	fbWriteSPLuxLevel				: SH_Light.FB_TwoVal_SelectOne_RTrigChange;
	fbWritePirDelayTIme			: SH_Light.FB_TwoVal_SelectOne_RTrigChange;
	stRoomDataPLC					: SH_Light.ST_RoomDataPLC	:=	(
																	uiPirOffDelayTime	:= 30,
																	uiSpLuxLevel			:= 500,
																	uiPirDimDelayTime	:= 15,
																	uiSpDimLuxLevel		:= 200);
																	
	fbBallastOnHours				: SH_Light.FB_CountOnHours;
	bEnableHourCount			: BOOL := TRUE;
	
	//Non-persistent modbus data
	bPirActive_MB				AT %MX40.0	: BOOL;				//bPirLys i gammel kode
	uiActLuxLevel_MB			AT %MB44	: UINT;				//intHMIAktueltLux i gammel kode
	uiActLightLevelPct_MB	    AT %MB52	: UINT;				//intDALI_Gruppe1_Lysniveau i gammel kode
	
	//For Conversion
	uiPirOffMinutes						: UINT;
	udTimeScaling						: UDINT := 60000;
	uiLuxOn								: UINT;
	
	//max values checks
	uiMaxLuxLevel						: UINT := 1023;
	uiMaxPirOffMinutes			    	: UINT := 180;

	
END_VAR

VAR CONSTANT
    Sensor_DALI_LINE_NUM				: BYTE := 3;
	DALI_LINE_NUM_LIGHT			    	: BYTE := 1;
	DALI_LINE_NUM_PENDANTS	            : BYTE := 1; //0=ingen pendler
	arrSensitivityOccupancy				: ARRAY[1..3] OF BYTE := [4,4,4];
END_VAR
VAR PERSISTENT
	stPirSensorData: SH_Light.ST_DALI_Sensor;
	stTuneData: SH_Light.ST_TuneData_EX;

	uiPirOffDelayTime_MB	AT %MB42	: UINT;				//ntHMI_Pir_SetValue i gammel kode
	uiSPLuxLevel_MB			AT %MB48	: UINT;				//intHMI_Lux_SetValue i gammel kode
	uiBallastOnHours_MB		AT %MB56	: UINT;				//dintHMILysbraendtimer1 i gammel kode
	byOnHoursOverflowCount				: BYTE;   
END_VAR

A_Buttons();
A_LightCtrl();
A_Sensor();
A_ModbusComm();

ACTION A_Buttons:
bTopButtonZone1		:= bTopButtonZone1_Visu;
bBottomButtonZone1	:= bBottomButtonZone1_Visu;
END_ACTION

ACTION A_LightCtrl:
bNeighborRoomsPir :=	P_Gang_2_446A.stPirSensorData.bPrc OR
									GVL_AHDataModbus.arrAH_NeighborRoomsPir[11][0] OR
									GVL_AHDataModbus.arrAH_NeighborRoomsPir[11][2] OR
									GVL_AHDataModbus.arrAH_NeighborRoomsPir[21][0] OR
									GVL_AHDataModbus.arrAH_NeighborRoomsPir[21][1];
									
fbLys(
	nZoneID:= 1, 
	bButtonZone1:= bTopButtonZone1, 
	bBottomButtonZone1 := bBottomButtonZone1,
	bButtonZone2:= bButtonZone2,
	bTopButtonOverride := (GVL_EnOcean.strEnOceanSwitch_AtriumNiveau_PladeB.bT2_ON OR GVL_EnOcean.strEnOceanSwitch_AtriumNiveau_Service.bT2_ON),
	bBottomButtonOverride := (GVL_EnOcean.strEnOceanSwitch_AtriumNiveau_PladeB.bT2_OFF OR GVL_EnOcean.strEnOceanSwitch_AtriumNiveau_Service.bT2_OFF),
	bNoButtons := TRUE,
	bNeighborRoomsPir	:=	bNeighborRoomsPir,
	fLuxOn:= fLuxOn, 
	fLuxDim:= fLuxDim, 
	tPIRDim:= tPIRDim, 
	tPIROff:= tPIROff, 
	fOffsetSec:= fOffsetSec, 
	bReInit:= , 
	stDaliSetup:= stDaliSetup, 
	ipCommunication_Prim:= P_DALI_Background.arrfbKL6821Communication[DALI_LINE_NUM_LIGHT], 
	//ipCommunication_Sec:= P_DALI_Background.arrfbKL6821Communication[DALI_LINE_NUM_LIGHT], 
	ipCommunication_Supl:= P_DALI_Background.arrfbKL6821Communication[DALI_LINE_NUM_PENDANTS], 
	fMinOutputPowerLevelRoom:= 15, 
	fMaxOutputPowerLevelRoom:= 100, 
	nCycleTimeInMS:= SH_Light.DALI_Param.nPlcTaskCycleTimeInMS*nDimCmdCycleTimeFactor , 
	bRunTuning:= bRunTuning, 
	bOccupiedRoom=> bOccupiedRoom, 
	bError_Prim=> , 
	nError_Prim=> , 
	stTuneData:=stTuneData , 
	stPirSensorData:= stPirSensorData, 
	stLiveData:= stLiveData);
END_ACTION

ACTION A_ModbusComm:
//Manage data for modbus communication

//Manage data for read-only in PLC
stRoomDataPLC.bPirActive			:= stPirSensorData.bPrc;
stRoomDataPLC.uiActLuxLevel			:= TO_UINT(TRUNC(stPirSensorData.fBrightness));
stRoomDataPLC.uiActLightLevelPct	:= TO_UINT(TRUNC(fbLys.fbBallast.fActlLgtLvl_Prim));
		//stRoomDataPLC.uiActLightLevelPct	:= TO_UINT(TRUNC(fbLys.fbBallast.fActlLgtLvl_Prim)); //if only one group light control
stRoomDataPLC.uiBallastOnHours		:= uiBallastOnHours_MB; //The calculation for BallastOnHours is stored directly to the MB register below


//Assign data for read-only to MB registers
bPirActive_MB			:= stRoomDataPLC.bPirActive;
uiActLuxLevel_MB		:= stRoomDataPLC.uiActLuxLevel;
uiActLightLevelPct_MB	:= stRoomDataPLC.uiActLightLevelPct;

	//calculate BallastOnHours
	fbBallastOnHours(
		bEnableHourCount	:= bEnableHourCount,
		bPauseCount			:= fbLys.fbLightCtrl.bOffZone1,
		uiOnHours			:= uiBallastOnHours_MB,			//OnHours is updated here
		byOverflowCount		:= byOnHoursOverflowCount);


//Manage data for read/write for both PLC and MB registers
fbWriteSPLuxLevel(	nMaxValOut	:= uiMaxLuxLevel,
					nValIn1		:= uiSPLuxLevel_MB,		//nValIn1 takes priotity in case of download or restart
					nValIn2		:= stRoomDataPLC.uiSpLuxLevel,
					nValOut		=> uiLuxOn
				);


fbWritePirDelayTIme(	nMaxValOut	:= uiMaxPirOffMinutes,
						nValIn1		:= uiPirOffDelayTime_MB,		//nValIn1 takes priotity in case of download or restart
						nValIn2		:= stRoomDataPLC.uiPirOffDelayTime,
						nValOut		=> uiPirOffMinutes
					);
					

//Convert read/write modbus data to appropriate datatypes in PLC
fLuxOn	:= TO_REAL(uiLuxOn);			
tPIROff	:= TO_TIME(uiPirOffMinutes*udTimeScaling); //Time conversion defaults to ms

fLuxDim	:= TO_REAL(stRoomDataPLC.uiSpDimLuxLevel);			
tPIRDim	:= TO_TIME(stRoomDataPLC.uiPirDimDelayTime*udTimeScaling); //Time conversion defaults to ms
END_ACTION

ACTION A_Sensor:

fbSensor.ipCommunication := P_DALI_Background.arrfbKL6821Communication[Sensor_DALI_LINE_NUM];

//only 1 sensor 
(*
fbSensor(
	byShrtAdr:= bySensorAddr,
	bInitialize:= bInitialize, 
	DALI_LINE_NUM:= Sensor_DALI_LINE_NUM, 
 	//bCancelHoldTimerOccupancy:= bCancelHoldTimerOccupancy, 
	stSensorSetup := stDaliSensorSetup,
	bInitErr=> bInitErr, 
	bInitDone=> bInitDone,
	stPirSensorData:= stPirSensorData, 
	arrSensorScales:= arrSensorScales);

*)
//several sensors	
fbSensor(
	arrShrtAdr:= arrSensorAddr,
	bInitialize:= bInitialize, 
	DALI_LINE_NUM:= Sensor_DALI_LINE_NUM, 
 	//bCancelHoldTimerOccupancy:= bCancelHoldTimerOccupancy, 
	stSensorSetup := stDaliSensorSetup,
	arrInitErr=> arrInitErr, 
	arrInitDone=> arrInitDone,
	stPirSensorData:= stPirSensorData, 
	arrSensorScales:= arrSensorScales);
END_ACTION

END_PROGRAM

// ---- POUs/Alle_Rum/Gange/Gang_2_446A/P_Gang_2_446A.TcPOU
PROGRAM P_Gang_2_446A
VAR

	fbLys		: FB_Light_Type_B;
	
	stDaliSetup	: SH_Light.ST_DALI_RoomSetup := (
														byShrtAdr_Prim := 54, 
														byGrpAdr_Prim := 1, 
														eMod_Prim := E_DALIAddressType.Group, 
														//byShrtAdr_Sec := 1, 
														//byGrpAdr_Sec := 1, 
														//eMod_Sec := E_DALIAddressType.Short, 
														//byShrtAdr_Supl := 1,
														//byGrpAdr_Supl := 1,
														//eMod_Prim := E_DALIAddressType.Short 
														DALI_LINE_NUM_PRIM := DALI_LINE_NUM_LIGHT, 
														DALI_LINE_NUM_SEC := 0, //0 = ingen zonestyring/vinduerække
														DALI_LINE_NUM_SUPL := DALI_LINE_NUM_PENDANTS);
														
	stLiveData				: SH_Light.ST_LiveData;
	bRunTuning					: BOOL;
	
	bTopButtonZone1				: BOOL;
	bTopButtonZone1_Visu		: BOOL;
	bBottomButtonZone1			: BOOL;
	bBottomButtonZone1_Visu	    : BOOL;
	bButtonZone2				: BOOL;
	bNeighborRoomsPir		    : BOOL;
	fLuxOn				     	: REAL;
	fLuxDim						: REAL;
	tPIRDim						: TIME;
	tPIROff						: TIME;
	fOffsetSec					: REAL := 20;
	bOccupiedRoom			    : BOOL;


// Sensor Settings
	fbSensor						: SH_Light.FB_NIKO_P46xx_1Pcs;
	//fbSensor						: SH_Light.FB_NIKO_P46xx_3Pcs;
	bySensorAddr				: BYTE := 63;
	//arrSensorAddr				: ARRAY[1..3] OF BYTE := [7,8,9];
	bInitialize						: BOOL := TRUE;
	stDaliSensorSetup			: ST_DALI_NIKOP46SetupData := (
																nSensitivityPIRSegmentA := arrSensitivityOccupancy[1],
																nSensitivityPIRSegmentB := arrSensitivityOccupancy[2],
																nSensitivityPIRSegmentC := arrSensitivityOccupancy[3]);
	bInitErr							: BOOL;
	bInitDone						: BOOL;
	//arrInitErr						: ARRAY [1..3] OF BOOL;
	//arrInitDone					: ARRAY [1..3] OF BOOL;
	arrSensorScales				: ARRAY [1..10] OF SH_Light.ST_DALI_SensorScaleMode := [
																						(fMeassureMaxSensor := rMeassure_Zone10, fReadMaxSensor := rRead_Zone10),																																										
																						9(())];
	bCancelHoldTimerOccupancy	: BOOL;
(*	eEventPriorityOccupancy		: E_DALIEventPriority := E_DALIEVENTPRIORITY.Middle;
	nHoldTimerOccupancy			: WORD := 5; // Value in s. 	
	nReportTimerOccupancy		: BYTE := 120; // Value in s, Preset manufacturer value
	nDeadtimeTimerOccupancy		: WORD := 100; // Value in ms, Predefined Value of DALI Standard
	bCancelHoldTimerOccupancy	: BOOL;
	nSensitivityOccupancy		: BYTE:= 3; //setting Sensivity (0..4) 0 (Off), 1 (Min), 2(Low), 3(High) and 4 (Max)

	bEnableLuxEvent				: BOOL;
	eEventPriorityBrightness	: E_DALIEventPriority := E_DALIEVENTPRIORITY.Middle;
	nDeadtimeTimerBrightness	: WORD := 1500; // Value in ms, Predefined Value of DALI Standard
	nHysteresisBrightness		: BYTE := 2; // Value in %
	nHysteresisMinBrightness	: BYTE := 10; // Absolute Value, depending on the manufacturer specific resolution
	nReportTimerBrightness		: BYTE := 120; // Value in s, Preset manufacturer value
*)

	//stDaliSetup: SH_Light.ST_DALI_RoomSetup
	//stRoomDataModbus			: SH_Light.ST_RoomDataModbus := ( bPirActive := bPirActive
	

	//ModbusComm setup
	
	fbWriteSPLuxLevel			: SH_Light.FB_TwoVal_SelectOne_RTrigChange;
	fbWritePirDelayTIme		: SH_Light.FB_TwoVal_SelectOne_RTrigChange;
	stRoomDataPLC				: SH_Light.ST_RoomDataPLC	:=	(
																	uiPirOffDelayTime	:= 30,
																	uiSpLuxLevel			:= 500,
																	uiPirDimDelayTime	:= 15,
																	uiSpDimLuxLevel		:= 200);
																	
	fbBallastOnHours				: SH_Light.FB_CountOnHours;
	bEnableHourCount			: BOOL := TRUE;
	
	//Non-persistent modbus data
	bPirActive_MB				AT %MX524.0	: BOOL;				//bPirLys i gammel kode
	uiActLuxLevel_MB			AT %MB528	: UINT;				//intHMIAktueltLux i gammel kode
	uiActLightLevelPct_MB	    AT %MB532	: UINT;				//intDALI_Gruppe1_Lysniveau i gammel kode
	
	//For Conversion
	uiPirOffMinutes						: UINT;
	udTimeScaling						: UDINT := 60000;
	uiLuxOn								: UINT;
	
	//max values checks
	uiMaxLuxLevel						: UINT := 1023;
	uiMaxPirOffMinutes				: UINT := 180;

	
END_VAR

VAR CONSTANT
    Sensor_DALI_LINE_NUM				: BYTE := 4;
	DALI_LINE_NUM_LIGHT			     	: BYTE := 4;
	DALI_LINE_NUM_PENDANTS	            : BYTE := 0; //0=ingen pendler	
	arrSensitivityOccupancy				: ARRAY[1..3] OF BYTE := [4,4,4];
END_VAR
VAR PERSISTENT
	stPirSensorData: SH_Light.ST_DALI_Sensor;
	stTuneData: SH_Light.ST_TuneData_EX;

	uiPirOffDelayTime_MB	AT %MB526	: UINT;				//ntHMI_Pir_SetValue i gammel kode
	uiSPLuxLevel_MB			AT %MB530	: UINT;				//intHMI_Lux_SetValue i gammel kode
	uiBallastOnHours_MB		AT %MB534	: UINT;				//dintHMILysbraendtimer1 i gammel kode
	byOnHoursOverflowCount				: BYTE;   
END_VAR

A_Buttons();
A_LightCtrl();
A_Sensor();
A_ModbusComm();

ACTION A_Buttons:
bTopButtonZone1		:= bTopButtonZone1_Visu;
bBottomButtonZone1	:= bBottomButtonZone1_Visu;
END_ACTION

ACTION A_LightCtrl:
bNeighborRoomsPir	:= 0;
fbLys(
	nZoneID:= 1, 
	bButtonZone1:= bTopButtonZone1,
	bBottomButtonZone1 := bBottomButtonZone1, 
	//bButtonZone2:= bButtonZone2,
	bNeighborRoomsPir := bNeighborRoomsPir,
	fLuxOn:= fLuxOn, 
	fLuxDim:= fLuxDim, 
	tPIRDim:= tPIRDim, 
	tPIROff:= tPIROff, 
	fOffsetSec:= fOffsetSec, 
	bReInit:= , 
	stDaliSetup:= stDaliSetup, 
	ipCommunication_Prim:= P_DALI_Background.arrfbKL6821Communication[DALI_LINE_NUM_LIGHT], 
	//ipCommunication_Sec:= P_DALI_Background.arrfbKL6821Communication[DALI_LINE_NUM_LIGHT], 
	//ipCommunication_Supl:= P_DALI_Background.arrfbKL6821Communication[DALI_LINE_NUM_PENDANTS], 
	fMinOutputPowerLevelRoom:= 15, 
	fMaxOutputPowerLevelRoom:= 100, 
	nCycleTimeInMS:= SH_Light.DALI_Param.nPlcTaskCycleTimeInMS*nDimCmdCycleTimeFactor , 
	bRunTuning:= bRunTuning, 
	bOccupiedRoom=> bOccupiedRoom, 
	bError_Prim=> , 
	nError_Prim=> , 
	stTuneData:=stTuneData , 
	stPirSensorData:= stPirSensorData, 
	stLiveData:= stLiveData);
END_ACTION

ACTION A_ModbusComm:
//Manage data for modbus communication

//Manage data for read-only in PLC
stRoomDataPLC.bPirActive			:= stPirSensorData.bPrc;
stRoomDataPLC.uiActLuxLevel			:= TO_UINT(TRUNC(stPirSensorData.fBrightness));
stRoomDataPLC.uiActLightLevelPct	:= TO_UINT(TRUNC(fbLys.fbBallast.fActlLgtLvl_Prim));
		//stRoomDataPLC.uiActLightLevelPct	:= TO_UINT(TRUNC(fbLys.fbBallast.fActlLgtLvl_Prim)); //if only one group light control
stRoomDataPLC.uiBallastOnHours		:= uiBallastOnHours_MB; //The calculation for BallastOnHours is stored directly to the MB register below


//Assign data for read-only to MB registers
bPirActive_MB			:= stRoomDataPLC.bPirActive;
uiActLuxLevel_MB		:= stRoomDataPLC.uiActLuxLevel;
uiActLightLevelPct_MB	:= stRoomDataPLC.uiActLightLevelPct;

	//calculate BallastOnHours
	fbBallastOnHours(
		bEnableHourCount	:= bEnableHourCount,
		bPauseCount			:= fbLys.fbLightCtrl.bOffZone1,
		uiOnHours			:= uiBallastOnHours_MB,			//OnHours is updated here
		byOverflowCount		:= byOnHoursOverflowCount);


//Manage data for read/write for both PLC and MB registers
fbWriteSPLuxLevel(	nMaxValOut	:= uiMaxLuxLevel,
					nValIn1		:= uiSPLuxLevel_MB,		//nValIn1 takes priotity in case of download or restart
					nValIn2		:= stRoomDataPLC.uiSpLuxLevel,
					nValOut		=> uiLuxOn
				);


fbWritePirDelayTIme(	nMaxValOut	:= uiMaxPirOffMinutes,
						nValIn1		:= uiPirOffDelayTime_MB,		//nValIn1 takes priotity in case of download or restart
						nValIn2		:= stRoomDataPLC.uiPirOffDelayTime,
						nValOut		=> uiPirOffMinutes
					);
					

//Convert read/write modbus data to appropriate datatypes in PLC
fLuxOn	:= TO_REAL(uiLuxOn);			
tPIROff	:= TO_TIME(uiPirOffMinutes*udTimeScaling); //Time conversion defaults to ms

fLuxDim	:= TO_REAL(stRoomDataPLC.uiSpDimLuxLevel);			
tPIRDim	:= TO_TIME(stRoomDataPLC.uiPirDimDelayTime*udTimeScaling); //Time conversion defaults to ms
END_ACTION

ACTION A_Sensor:

fbSensor.ipCommunication := P_DALI_Background.arrfbKL6821Communication[Sensor_DALI_LINE_NUM];

//only 1 sensor
fbSensor(
	byShrtAdr:= bySensorAddr,
	bInitialize:= bInitialize, 
	DALI_LINE_NUM:= Sensor_DALI_LINE_NUM, 
 	//bCancelHoldTimerOccupancy:= bCancelHoldTimerOccupancy, 
	stSensorSetup := stDaliSensorSetup,
	bInitErr=> bInitErr, 
	bInitDone=> bInitDone,
	stPirSensorData:= stPirSensorData, 
	arrSensorScales:= arrSensorScales);


(*//several sensors	
fbSensor(
	arrShrtAdr:= arrSensorAddr,
	bInitialize:= bInitialize, 
	DALI_LINE_NUM:= Sensor_DALI_LINE_NUM, 
 	//bCancelHoldTimerOccupancy:= bCancelHoldTimerOccupancy, 
	stSensorSetup := stDaliSensorSetup,
	arrInitErr=> arrInitErr, 
	arrInitDone=> arrInitDone,
	stPirSensorData:= stPirSensorData, 
	arrSensorScales:= arrSensorScales);
	*)
END_ACTION

END_PROGRAM

// ---- POUs/DALI/DALI_Setup/FBs/FB_Part103Addressing.TcPOU
FUNCTION_BLOCK FB_Part103Addressing
VAR_INPUT
	ipDALICommunication			:	I_DALICommunication;
END_VAR
VAR_OUTPUT
	bBusy						:	BOOL;
END_VAR
VAR
	{region "Visu"}
	bScanDevices				:	BOOL;
	bStartChangeAddress			:	BOOL;
	bStartRandomAddressing		:	BOOL;
	nStartAddress				:	BYTE;
	bNewInstallation			:	BOOL;
	bOpticalFeedback			:	BOOL;
	bHideWaitSymbol				:	BOOL := TRUE;
	{endregion}
	nStep						:	INT;
	nAddress					:	INT;
	aChangeAddressList			:	ARRAY [0..63] OF ST_DALIChangeAddressList;
	aShortAddress				:	ARRAY [0..63] OF INT;
	aNoShortAddress				:	ARRAY [0..63] OF BOOL;
	nRow						:	INT;
	nHideLine					:	INT; // Variable to find out how many rows are used

	fb103StartQuiescentMode		:	FB_DALI103StartQuiescentMode(0);
	fb103StopQuiescentMode		:	FB_DALI103StopQuiescentMode(0);
	fb103Addressing				:	FB_DALI103Addressing(0);
	fb103QueryRandomAddress		:	FB_DALI103QueryRandomAddress(0);
	fb103ChangeAddresses		:	FB_DALI103ChangeAddresses(0);
END_VAR

{region "Detect Commands"}
IF (bStartRandomAddressing AND (nStep = 0)) THEN
	nStep := 5;
	bStartRandomAddressing := FALSE;
	bHideWaitSymbol := FALSE;
END_IF

IF (bScanDevices AND (nStep = 0)) THEN
	nStep := 20;
	nAddress :=0;
	bScanDevices := FALSE;
	bHideWaitSymbol := FALSE;
END_IF

IF (bStartChangeAddress AND (nStep = 0)) THEN
	nStep := 60;
	bStartChangeAddress := FALSE;
	bHideWaitSymbol := FALSE;
END_IF
{endregion}
{region "Manage Dialog Selection}
IF (nStep = 0) THEN
	bBusy := FALSE;
ELSE
	bBusy := TRUE;
END_IF
{endregion}	 
{region "Execute Commands"}
CASE nStep OF
0:
{region "Init"}
	bScanDevices := FALSE;
	bStartChangeAddress := FALSE;
	bStartRandomAddressing := FALSE;
	bHideWaitSymbol := TRUE;

	fb103StartQuiescentMode.ipDALICommunication := ipDALICommunication;
	fb103StopQuiescentMode.ipDALICommunication := ipDALICommunication;
	fb103Addressing.ipDALICommunication := ipDALICommunication;
	fb103QueryRandomAddress.ipDALICommunication := ipDALICommunication;
	fb103ChangeAddresses.ipDALICommunication := ipDALICommunication;
{endregion}
5:
{region "Start Qiescent Mode"}
	fb103StartQuiescentMode(bStart := TRUE,
							eAddressType := Tc3_DALI.E_DALIAddressType.Broadcast,
							eCommandPriority := Tc3_DALI.E_DALICommandPriority.Middle);
	IF (NOT fb103StartQuiescentMode.bBusy) THEN
		fb103StartQuiescentMode(bStart:= FALSE);
		nStep := 10;
	END_IF
{endregion}
10:
{region "RandomAddressing"}
	IF bNewInstallation THEN
		fb103Addressing.nOptions := Tc3_DALI.GVL.cCompleteNewInstallation;
	END_IF

	IF bOpticalFeedback THEN
		fb103Addressing.nOptions := Tc3_DALI.GVL.cOpticalFeedback;
	END_IF

	IF bNewInstallation AND bOpticalFeedback THEN
		fb103Addressing.nOptions := Tc3_DALI.GVL.cCompleteNewInstallation OR Tc3_DALI.GVL.cOpticalFeedback;
	END_IF
	fb103Addressing(bStart := TRUE,
					nStartWithShortAddress := nStartAddress);
	IF (NOT fb103Addressing.bBusy) THEN
		fb103Addressing(bStart := FALSE);
		nStep := 15;
	END_IF
{endregion}
15:
{region "Stop Qiescent Mode"}
	fb103StopQuiescentMode(	bStart := TRUE,
							eAddressType := Tc3_DALI.E_DALIAddressType.Broadcast,
							eCommandPriority := Tc3_DALI.E_DALICommandPriority.Middle);
	IF (NOT fb103StopQuiescentMode.bBusy) THEN
		fb103StopQuiescentMode(	bStart:= FALSE);
		nStep := 0;
	END_IF
{endregion}
{region "Read Existing Addresses"}
20:
{region "Start Qiescent Mode"}
	fb103StartQuiescentMode(bStart := TRUE,
							eAddressType := Tc3_DALI.E_DALIAddressType.Broadcast,
							eCommandPriority := Tc3_DALI.E_DALICommandPriority.Middle);
	IF (NOT fb103StartQuiescentMode.bBusy) THEN
		fb103StartQuiescentMode(bStart:= FALSE);
		nStep := 30;
	END_IF
{endregion}
30:
	// Query of the new random addresses to find out which short addresses are existing.
	fb103QueryRandomAddress (	bStart := TRUE,
								nAddress := TO_BYTE(nAddress),
								eAddressType := Tc3_DALI.E_DALIAddressType.Short,
								nRandomAddress => aChangeAddressList[nAddress].nRandomAddress);
	IF (NOT fb103QueryRandomAddress.bBusy) THEN
		fb103QueryRandomAddress(bStart := FALSE);
		nAddress := nAddress + 1;
		IF (nAddress > 63) THEN
			nStep := 40;
		END_IF
	END_IF
40:
	// Write the existing short addresses into the table 
	nRow := 0;
	FOR nAddress := 0 TO 63 DO
		IF (aChangeAddressList[nAddress].nRandomAddress > 0) THEN
			aChangeAddressList[nRow].nOldAddress := TO_BYTE(nAddress);
			nRow := nRow + 1;
		END_IF
	END_FOR
	nStep := 50;
50:
	// Hide unused rows in the table
	nHideLine := 0;
	FOR nAddress := 0 TO 63 DO 
		IF (aChangeAddressList[nAddress].nRandomAddress <> 0) THEN
			aShortAddress[nHideLine] := nAddress;
			nHideLine := nHideLine + 1;
		END_IF
	END_FOR
	FOR nAddress := nHideLine TO 63 DO 
		aNoShortAddress[nAddress] := TRUE;
	END_FOR
	FOR nAddress := 0 TO (nHideLine - 1) DO
		aNoShortAddress[nAddress] := FALSE;
	END_FOR
	aChangeAddressList[nHideLine].nOldAddress := 255;
	FOR nAddress := 0 TO nHideLine DO
		aChangeAddressList[nAddress].nNewAddress := aChangeAddressList[nAddress].nOldAddress;
	END_FOR
	nStep := 55;
{endregion}
55:
{region "Stop Qiescent Mode"}
	fb103StopQuiescentMode(	bStart := TRUE,
							eAddressType := Tc3_DALI.E_DALIAddressType.Broadcast,
							eCommandPriority := Tc3_DALI.E_DALICommandPriority.Middle);
	IF (NOT fb103StopQuiescentMode.bBusy) THEN
		fb103StopQuiescentMode(	bStart:= FALSE);
		nStep := 0;
	END_IF
{endregion}
60:
{region "Write Changed Addresses}
	fb103ChangeAddresses(	bStart := TRUE,
							aChangeAddressList := aChangeAddressList);
	IF (NOT fb103ChangeAddresses.bBusy) THEN
		fb103ChangeAddresses(	bStart := FALSE,
								aChangeAddressList := aChangeAddressList);
		nStep := 70;
	END_IF
{endregion}
70:
{region "Write New Address To Old Address}
	FOR nAddress := 0 TO 63 DO
		aChangeAddressList[nAddress].nOldAddress := aChangeAddressList[nAddress].nNewAddress;
	END_FOR
	nStep := 0;
{endregion}
END_CASE

END_FUNCTION_BLOCK

// ---- POUs/EnOcean/P_EnOcean.TcPOU
PROGRAM P_EnOcean
VAR
	fbKL6581			: FB_KL6581;
	stKL6581_in  AT %I* : KL6581_INPUT;
	stKL6581_out AT %Q*	: KL6581_OUTPUT;
	stKL6581			: STR_KL6581;
	bInitCom			: BOOL := TRUE;
	
	arrEnOcean_Search	: ARRAY [1..8] OF FB_EnOcean_Search;
	nSearchIdx			: BYTE;
	bSerach				: BOOL;
	arrDevices			: ARRAY [1..8] OF INT;
	arrID				: ARRAY [1..8, 0..255] OF DWORD;
	
		//Trykknapper Atrium
	fbAtriumNiveau_Tryk_PladeB				: FB_Rec_RPS_Switch;
	fbAtriumNiveau_Tryk_Sevice				: FB_Rec_RPS_Switch;			

	//Trykknapper på gange

	
	//Trykknapper i rum
	fbRum_1_421_Tryk						: FB_Rec_RPS_Switch;
	fbRum_1_422_Tryk						: FB_Rec_RPS_Switch;
	fbRum_1_424_Tryk						: FB_Rec_RPS_Switch;
    fbRum_1_425_Tryk						: FB_Rec_RPS_Switch;
    fbRum_1_427_Tryk						: FB_Rec_RPS_Switch;
    fbRum_1_428_Tryk						: FB_Rec_RPS_Switch; 
    fbRum_1_429_Tryk						: FB_Rec_RPS_Switch;
    fbRum_1_430_Tryk						: FB_Rec_RPS_Switch;
    fbRum_1_431_Tryk						: FB_Rec_RPS_Switch;
    fbRum_1_432_Tryk						: FB_Rec_RPS_Switch;
    fbRum_1_433_Tryk						: FB_Rec_RPS_Switch;
    fbRum_1_434_Tryk						: FB_Rec_RPS_Switch;
    fbRum_1_435_Tryk						: FB_Rec_RPS_Switch;

    fbRum_Kantine_Tryk						: FB_Rec_RPS_Switch;
END_VAR

VAR CONSTANT
	byNode_1: BYTE := 1;
	byNode_2: BYTE := 2;
	byNode_3: BYTE := 3;
	byNode_4: BYTE := 4;
	byNode_5: BYTE := 5;
	byNode_6: BYTE := 6;
	byNode_7: BYTE := 7;
	byNode_8: BYTE := 8;
END_VAR


(* Kommunikation mit der KL6581. *)
(* Communication with the KL6581. *)
fbKL6581(
	bInit			:= bInitCom,
	nIdx			:= 2,
	stKL6581_in		:= stKL6581_In,
	stKL6581_out	:= stKL6581_Out,
	bReady			=> ,
	bBusy			=> ,
	bError			=> ,
	iErrorID		=> ,
	str_KL6581		=> stKL6581);

GVL_AHDataModbus.EnOceanError	:= TO_UINT(fbKL6581.iErrorID);
(* Warten bis der Kommunikationsbaustein initialisiert wurde.*)
(* Wait until the communication function block has been initialized. *)
IF (NOT fbKL6581.bReady) THEN
	RETURN;
END_IF

FOR nSearchIdx:= 1 TO 8 DO
	arrEnOcean_Search[nSearchIdx](
		bStart:= TRUE, 
		str_KL6581:= stKL6581 , 
		byNode:= nSearchIdx, 
		bReceive=> , 
		iDevices=>arrDevices[nSearchIdx] , 
		ar_ID=> );
		
		MEMCPY(ADR(arrID[nSearchIdx,0]), ADR(arrEnOcean_Search[nSearchIdx].ar_ID), SIZEOF(arrEnOcean_Search[nSearchIdx].ar_ID)); 
END_FOR

//Gange



//RUM
 //
 
 
A_rum_1_421(); 
A_rum_1_422();
A_rum_1_424(); 
A_rum_1_425();
A_Rum_1_427();
A_Rum_1_428();
A_Rum_1_429();
A_Rum_1_430();

A_Rum_1_435();
A_Rum_1_434(); 
A_Rum_1_433();
A_Rum_1_432();
A_Rum_1_431();



//AtriumNiveau
A_AtriumNiveau();

ACTION A_AtriumNiveau:
fbAtriumNiveau_Tryk_PladeB(
	str_KL6581:=stKL6581 , 
	byNode:=2, 
	dw_ID:= 16#0029B92D, 
	str_EnOceanSwitch=> GVL_EnOcean.strEnOceanSwitch_AtriumNiveau_PladeB,
	by_Node=> , 
	bReceive=> );

//knap 2 
(*
fbAtriumNiveau_Tryk_Sevice(
	str_KL6581:=stKL6581 , 
	byNode:=0, 
	dw_ID:= 16#00FEE4FE87, 
	str_EnOceanSwitch=> GVL_EnOcean.strEnOceanSwitch_AtriumNiveau_Service, 
	by_Node=> , 
	bReceive=> );
*)
END_ACTION

ACTION A_Rum_1_421:
fbRum_1_421_Tryk(
	str_KL6581:=stKL6581 , 
	byNode:=4 , 
	dw_ID:= 16#002E7C21, 
	str_EnOceanSwitch=> GVL_EnOcean.strEnOceanSwitch_Rum_1_421, 
	by_Node=> , 
	bReceive=> );
END_ACTION

ACTION A_Rum_1_422:
fbRum_1_422_Tryk(
	str_KL6581:=stKL6581 , 
	byNode:=4 , 
	dw_ID:= 16#002F6679, 
	str_EnOceanSwitch=> GVL_EnOcean.strEnOceanSwitch_Rum_1_422, 
	by_Node=> , 
	bReceive=> );
END_ACTION

ACTION A_Rum_1_424:
fbRum_1_424_Tryk(
	str_KL6581:=stKL6581 , 
	byNode:=4 , 
	dw_ID:= 16#002F3103, 
	str_EnOceanSwitch=> GVL_EnOcean.strEnOceanSwitch_Rum_1_424, 
	by_Node=> , 
	bReceive=> );
END_ACTION

ACTION A_Rum_1_425:
fbRum_1_425_Tryk(
	str_KL6581:=stKL6581 , 
	byNode:=4 , 
	dw_ID:= 16#002E7C18, 
	str_EnOceanSwitch=> GVL_EnOcean.strEnOceanSwitch_Rum_1_425, 
	by_Node=> , 
	bReceive=> );
END_ACTION

ACTION A_Rum_1_427:
fbRum_1_427_Tryk(
	str_KL6581:=stKL6581 , 
	byNode:=4 , 
	dw_ID:= 16#00336F5B, 
	str_EnOceanSwitch=> GVL_EnOcean.strEnOceanSwitch_Rum_1_427, 
	by_Node=> , 
	bReceive=> );
END_ACTION

ACTION A_Rum_1_428:
fbRum_1_428_Tryk(
	str_KL6581:=stKL6581 , 
	byNode:=4 , 
	dw_ID:= 16#0029B882, 
	str_EnOceanSwitch=> GVL_EnOcean.strEnOceanSwitch_Rum_1_428, 
	by_Node=> , 
	bReceive=> );
END_ACTION

ACTION A_Rum_1_429:
fbRum_1_429_Tryk(
	str_KL6581:=stKL6581 , 
	byNode:=4 , 
	dw_ID:= 16#00336F68, 
	str_EnOceanSwitch=> GVL_EnOcean.strEnOceanSwitch_Rum_1_429, 
	by_Node=> , 
	bReceive=> );
END_ACTION

ACTION A_Rum_1_430:
fbRum_1_430_Tryk(
	str_KL6581:=stKL6581 , 
	byNode:=4 , 
	dw_ID:= 16#00336F55, 
	str_EnOceanSwitch=> GVL_EnOcean.strEnOceanSwitch_Rum_1_430, 
	by_Node=> , 
	bReceive=> );
END_ACTION

ACTION A_Rum_1_431:
fbRum_1_431_Tryk(
	str_KL6581:=stKL6581 , 
	byNode:=2 , 
	dw_ID:= 16#00336F51, 
	str_EnOceanSwitch=> GVL_EnOcean.strEnOceanSwitch_Rum_1_431, 
	by_Node=> , 
	bReceive=> );
END_ACTION

ACTION A_Rum_1_432:
fbRum_1_432_Tryk(
	str_KL6581:=stKL6581 , 
	byNode:=2 , 
	dw_ID:= 16#00336F65, 
	str_EnOceanSwitch=> GVL_EnOcean.strEnOceanSwitch_Rum_1_432, 
	by_Node=> , 
	bReceive=> );
END_ACTION

ACTION A_Rum_1_433:
fbRum_1_433_Tryk(
	str_KL6581:=stKL6581 , 
	byNode:=4 , 
	dw_ID:= 16#00336F66, 
	str_EnOceanSwitch=> GVL_EnOcean.strEnOceanSwitch_Rum_1_433, 
	by_Node=> , 
	bReceive=> );
END_ACTION

ACTION A_Rum_1_434:
fbRum_1_434_Tryk(
	str_KL6581:=stKL6581 , 
	byNode:=2 , 
	dw_ID:= 16#00336F4B, 
	str_EnOceanSwitch=> GVL_EnOcean.strEnOceanSwitch_Rum_1_434, 
	by_Node=> , 
	bReceive=> );
END_ACTION

ACTION A_Rum_1_435:
fbRum_1_435_Tryk(
	str_KL6581:=stKL6581 , 
	byNode:=2 , 
	dw_ID:= 16#0029AADA, 
	str_EnOceanSwitch=> GVL_EnOcean.strEnOceanSwitch_Rum_1_435, 
	by_Node=> , 
	bReceive=> );
END_ACTION

END_PROGRAM

// ---- POUs/MAIN.TcPOU
PROGRAM MAIN
VAR
	nAlive: INT;
	breset: BOOL;
	nDemoVariable : INT;
	nCX8200_State	AT %I*	: UINT;
END_VAR

VAR PERSISTENT
	nDemoVar_Persist: INT;
END_VAR

nAlive:= nAlive + 1;
GVL_AHDataModbus.nCX8200_State_MB := nCX8200_State;

P_SystemDK.M_nCyclic(bReset := breset );
P_DALI_DIAG();
DALI_Commissioning();
P_DALI_Energy_Line();
P_AHModbusComm();


//Gange
P_Gang_1_418();
P_Gang_1_417();
P_Gang_1_426();
P_Gang_2_446A();
P_Gang_7_401();

//Rum
P_Rum_1_435();
P_Rum_1_434();
P_Rum_1_433();
P_Rum_1_432();
P_Rum_1_431();
P_Rum_1_430();
P_Rum_1_429();
P_Rum_1_428();
P_Rum_1_427();

P_Rum_1_425();
P_Rum_1_424();
P_Rum_1_422();
P_Rum_1_421();


//Testprogrammer
//P_DALI_Energy_Firmware_Test();

END_PROGRAM

// ---- POUs/Alle_Rum/Gange/Gang_1_147/Visualization_4_330_2_1.TcVIS
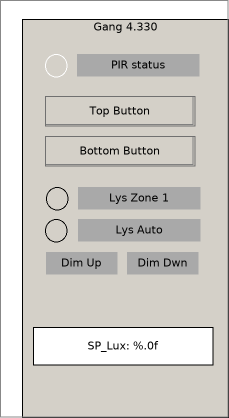
VISUALIZATION Visualization_4_330_2_1  // 229x418
    RoundedRectangle (22,19 207x399), "Gang 4.330"
    Rectangle (33,327 180x38), "SP_Lux: %.0f", text variable: P_Gang_2_143A.arrfbLysGruppe[1].fbLightCtrl.fLuxZone1
    Button (45,96 150x30), "Top Button"
        tap P_Gang_2_143A.bTopButtonZone1_Visu
    Button (45,136 150x30), "Bottom Button"
        tap P_Gang_2_143A.bBottomButtonZone1_Visu
    Ellipse (46,187 22x23), colour toggle: P_Gang_2_143A.fbLys.fbLightCtrl.bOnZone1
    Rectangle (78,187 122x22), "Lys Zone 1"
    Rectangle (46,252 71x22), "Dim Up", colour toggle: P_Gang_2_143A.arrfbLysGruppe[1].fbLightCtrl.bDimUp
    Rectangle (127,252 71x22), "Dim Dwn", colour toggle: P_Gang_2_143A.arrfbLysGruppe[1].fbLightCtrl.bDimDwn
    Ellipse (45,219 22x23), colour toggle: P_Gang_2_143A.arrfbLysGruppe[1].fbLightCtrl.bAutoZone1
    Rectangle (78,219 122x22), "Lys Auto"
    Ellipse (45,54 22x23), colour toggle: P_Gang_2_143A.arrfbLysGruppe[1].fbLightCtrl.bPIR
    Rectangle (77,54 122x22), "PIR status"
END_VISUALIZATION

// ---- POUs/Alle_Rum/Rum_Med_DALI_Pir/Rum_1_421/Visualization_4_330_1_1_1_1_2_1_1_1_1.TcVIS
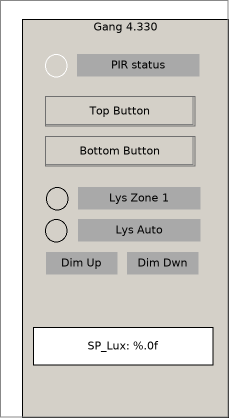
VISUALIZATION Visualization_4_330_1_1_1_1_2_1_1_1_1  // 229x418
    RoundedRectangle (22,19 207x399), "Gang 4.330"
    Rectangle (33,327 180x38), "SP_Lux: %.0f", text variable: P_Gang_5_135A.arrfbLysGruppe[1].fbLightCtrl.fLuxZone1
    Button (45,96 150x30), "Top Button"
        tap P_Gang_5_135A.bTopButtonZone1_Visu
    Button (45,136 150x30), "Bottom Button"
        tap P_Gang_5_135A.bBottomButtonZone1_Visu
    Ellipse (46,187 22x23), colour toggle: P_Gang_5_135A.fbLys.fbLightCtrl.bOnZone1
    Rectangle (78,187 122x22), "Lys Zone 1"
    Rectangle (46,252 71x22), "Dim Up", colour toggle: P_Gang_5_135A.arrfbLysGruppe[1].fbLightCtrl.bDimUp
    Rectangle (127,252 71x22), "Dim Dwn", colour toggle: P_Gang_5_135A.arrfbLysGruppe[1].fbLightCtrl.bDimDwn
    Ellipse (45,219 22x23), colour toggle: P_Gang_5_135A.arrfbLysGruppe[1].fbLightCtrl.bAutoZone1
    Rectangle (78,219 122x22), "Lys Auto"
    Ellipse (45,54 22x23), colour toggle: P_Gang_5_135A.arrfbLysGruppe[1].fbLightCtrl.bPIR
    Rectangle (77,54 122x22), "PIR status"
END_VISUALIZATION

// ---- POUs/Alle_Rum/Rum_Med_DALI_Pir/Rum_1_422/Visualization_4_330_1_1_1_1_2_1_1_1.TcVIS
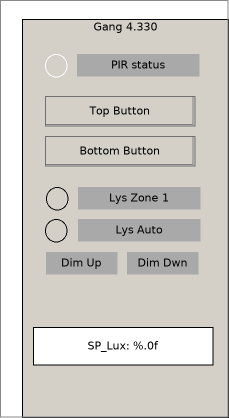
VISUALIZATION Visualization_4_330_1_1_1_1_2_1_1_1  // 229x418
    RoundedRectangle (22,19 207x399), "Gang 4.330"
    Rectangle (33,327 180x38), "SP_Lux: %.0f", text variable: P_Gang_5_135A.arrfbLysGruppe[1].fbLightCtrl.fLuxZone1
    Button (45,96 150x30), "Top Button"
        tap P_Gang_5_135A.bTopButtonZone1_Visu
    Button (45,136 150x30), "Bottom Button"
        tap P_Gang_5_135A.bBottomButtonZone1_Visu
    Ellipse (46,187 22x23), colour toggle: P_Gang_5_135A.fbLys.fbLightCtrl.bOnZone1
    Rectangle (78,187 122x22), "Lys Zone 1"
    Rectangle (46,252 71x22), "Dim Up", colour toggle: P_Gang_5_135A.arrfbLysGruppe[1].fbLightCtrl.bDimUp
    Rectangle (127,252 71x22), "Dim Dwn", colour toggle: P_Gang_5_135A.arrfbLysGruppe[1].fbLightCtrl.bDimDwn
    Ellipse (45,219 22x23), colour toggle: P_Gang_5_135A.arrfbLysGruppe[1].fbLightCtrl.bAutoZone1
    Rectangle (78,219 122x22), "Lys Auto"
    Ellipse (45,54 22x23), colour toggle: P_Gang_5_135A.arrfbLysGruppe[1].fbLightCtrl.bPIR
    Rectangle (77,54 122x22), "PIR status"
END_VISUALIZATION

// ---- POUs/Alle_Rum/Rum_Med_DALI_Pir/Rum_1_427/Visualization_5_338_1_1_1_1_2_1_1_1_1.TcVIS
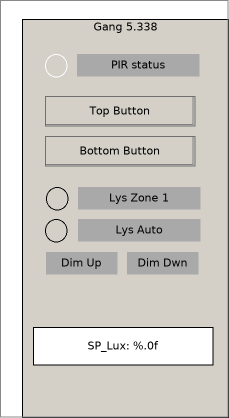
VISUALIZATION Visualization_5_338_1_1_1_1_2_1_1_1_1  // 229x418
    RoundedRectangle (22,19 207x399), "Gang 5.338"
    Rectangle (33,327 180x38), "SP_Lux: %.0f", text variable: P_Gang_5_338.arrfbLysGruppe[1].fbLightCtrl.fLuxZone1
    Button (45,96 150x30), "Top Button"
        tap P_Gang_5_338.bTopButtonZone1_Visu
    Button (45,136 150x30), "Bottom Button"
        tap P_Gang_5_338.bBottomButtonZone1_Visu
    Ellipse (46,187 22x23), colour toggle: P_Gang_5_338.arrfbLysGruppe[1].fbLightCtrl.bOnZone1
    Rectangle (78,187 122x22), "Lys Zone 1"
    Rectangle (46,252 71x22), "Dim Up", colour toggle: P_Gang_5_338.arrfbLysGruppe[1].fbLightCtrl.bDimUp
    Rectangle (127,252 71x22), "Dim Dwn", colour toggle: P_Gang_5_338.arrfbLysGruppe[1].fbLightCtrl.bDimDwn
    Ellipse (45,219 22x23), colour toggle: P_Gang_5_338.arrfbLysGruppe[1].fbLightCtrl.bAutoZone1
    Rectangle (78,219 122x22), "Lys Auto"
    Ellipse (45,54 22x23), colour toggle: P_Gang_5_338.arrfbLysGruppe[1].fbLightCtrl.bPIR
    Rectangle (77,54 122x22), "PIR status"
END_VISUALIZATION

// ---- POUs/Alle_Rum/Rum_Med_DALI_Pir/Rum_1_430/Visualization_5_338_1_1_1_1_2_1.TcVIS
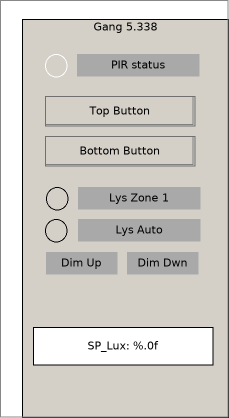
VISUALIZATION Visualization_5_338_1_1_1_1_2_1  // 229x418
    RoundedRectangle (22,19 207x399), "Gang 5.338"
    Rectangle (33,327 180x38), "SP_Lux: %.0f", text variable: P_Gang_5_338.arrfbLysGruppe[1].fbLightCtrl.fLuxZone1
    Button (45,96 150x30), "Top Button"
        tap P_Gang_5_338.bTopButtonZone1_Visu
    Button (45,136 150x30), "Bottom Button"
        tap P_Gang_5_338.bBottomButtonZone1_Visu
    Ellipse (46,187 22x23), colour toggle: P_Gang_5_338.arrfbLysGruppe[1].fbLightCtrl.bOnZone1
    Rectangle (78,187 122x22), "Lys Zone 1"
    Rectangle (46,252 71x22), "Dim Up", colour toggle: P_Gang_5_338.arrfbLysGruppe[1].fbLightCtrl.bDimUp
    Rectangle (127,252 71x22), "Dim Dwn", colour toggle: P_Gang_5_338.arrfbLysGruppe[1].fbLightCtrl.bDimDwn
    Ellipse (45,219 22x23), colour toggle: P_Gang_5_338.arrfbLysGruppe[1].fbLightCtrl.bAutoZone1
    Rectangle (78,219 122x22), "Lys Auto"
    Ellipse (45,54 22x23), colour toggle: P_Gang_5_338.arrfbLysGruppe[1].fbLightCtrl.bPIR
    Rectangle (77,54 122x22), "PIR status"
END_VISUALIZATION

// ---- POUs/Alle_Rum/Rum_Med_DALI_Pir/Rum_1_429/Visualization_5_338_1_1_1_1_2_1_1.TcVIS
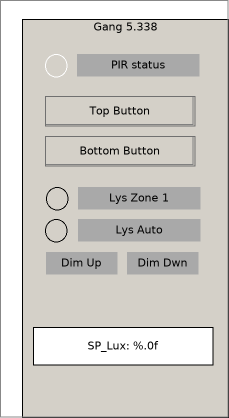
VISUALIZATION Visualization_5_338_1_1_1_1_2_1_1  // 229x418
    RoundedRectangle (22,19 207x399), "Gang 5.338"
    Rectangle (33,327 180x38), "SP_Lux: %.0f", text variable: P_Gang_5_338.arrfbLysGruppe[1].fbLightCtrl.fLuxZone1
    Button (45,96 150x30), "Top Button"
        tap P_Gang_5_338.bTopButtonZone1_Visu
    Button (45,136 150x30), "Bottom Button"
        tap P_Gang_5_338.bBottomButtonZone1_Visu
    Ellipse (46,187 22x23), colour toggle: P_Gang_5_338.arrfbLysGruppe[1].fbLightCtrl.bOnZone1
    Rectangle (78,187 122x22), "Lys Zone 1"
    Rectangle (46,252 71x22), "Dim Up", colour toggle: P_Gang_5_338.arrfbLysGruppe[1].fbLightCtrl.bDimUp
    Rectangle (127,252 71x22), "Dim Dwn", colour toggle: P_Gang_5_338.arrfbLysGruppe[1].fbLightCtrl.bDimDwn
    Ellipse (45,219 22x23), colour toggle: P_Gang_5_338.arrfbLysGruppe[1].fbLightCtrl.bAutoZone1
    Rectangle (78,219 122x22), "Lys Auto"
    Ellipse (45,54 22x23), colour toggle: P_Gang_5_338.arrfbLysGruppe[1].fbLightCtrl.bPIR
    Rectangle (77,54 122x22), "PIR status"
END_VISUALIZATION

// ---- POUs/Alle_Rum/Rum_Med_DALI_Pir/Rum_1_432/Visualization_5_338_1_1_1_1_1.TcVIS
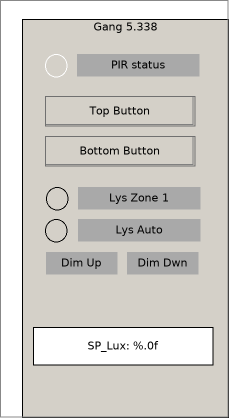
VISUALIZATION Visualization_5_338_1_1_1_1_1  // 229x418
    RoundedRectangle (22,19 207x399), "Gang 5.338"
    Rectangle (33,327 180x38), "SP_Lux: %.0f", text variable: P_Gang_5_338.arrfbLysGruppe[1].fbLightCtrl.fLuxZone1
    Button (45,96 150x30), "Top Button"
        tap P_Gang_5_338.bTopButtonZone1_Visu
    Button (45,136 150x30), "Bottom Button"
        tap P_Gang_5_338.bBottomButtonZone1_Visu
    Ellipse (46,187 22x23), colour toggle: P_Gang_5_338.arrfbLysGruppe[1].fbLightCtrl.bOnZone1
    Rectangle (78,187 122x22), "Lys Zone 1"
    Rectangle (46,252 71x22), "Dim Up", colour toggle: P_Gang_5_338.arrfbLysGruppe[1].fbLightCtrl.bDimUp
    Rectangle (127,252 71x22), "Dim Dwn", colour toggle: P_Gang_5_338.arrfbLysGruppe[1].fbLightCtrl.bDimDwn
    Ellipse (45,219 22x23), colour toggle: P_Gang_5_338.arrfbLysGruppe[1].fbLightCtrl.bAutoZone1
    Rectangle (78,219 122x22), "Lys Auto"
    Ellipse (45,54 22x23), colour toggle: P_Gang_5_338.arrfbLysGruppe[1].fbLightCtrl.bPIR
    Rectangle (77,54 122x22), "PIR status"
END_VISUALIZATION

// ---- POUs/Alle_Rum/Rum_Med_DALI_Pir/Rum_1_431/Visualization_5_338_1_1_1_1_2.TcVIS
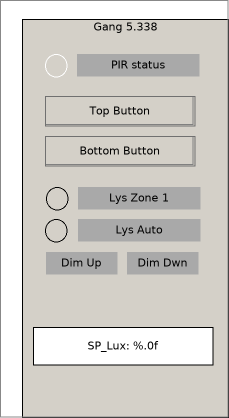
VISUALIZATION Visualization_5_338_1_1_1_1_2  // 229x418
    RoundedRectangle (22,19 207x399), "Gang 5.338"
    Rectangle (33,327 180x38), "SP_Lux: %.0f", text variable: P_Gang_5_338.arrfbLysGruppe[1].fbLightCtrl.fLuxZone1
    Button (45,96 150x30), "Top Button"
        tap P_Gang_5_338.bTopButtonZone1_Visu
    Button (45,136 150x30), "Bottom Button"
        tap P_Gang_5_338.bBottomButtonZone1_Visu
    Ellipse (46,187 22x23), colour toggle: P_Gang_5_338.arrfbLysGruppe[1].fbLightCtrl.bOnZone1
    Rectangle (78,187 122x22), "Lys Zone 1"
    Rectangle (46,252 71x22), "Dim Up", colour toggle: P_Gang_5_338.arrfbLysGruppe[1].fbLightCtrl.bDimUp
    Rectangle (127,252 71x22), "Dim Dwn", colour toggle: P_Gang_5_338.arrfbLysGruppe[1].fbLightCtrl.bDimDwn
    Ellipse (45,219 22x23), colour toggle: P_Gang_5_338.arrfbLysGruppe[1].fbLightCtrl.bAutoZone1
    Rectangle (78,219 122x22), "Lys Auto"
    Ellipse (45,54 22x23), colour toggle: P_Gang_5_338.arrfbLysGruppe[1].fbLightCtrl.bPIR
    Rectangle (77,54 122x22), "PIR status"
END_VISUALIZATION

// ---- POUs/Alle_Rum/Rum_Med_DALI_Pir/Rum_1_434/Visualization_5_338_1_1.TcVIS
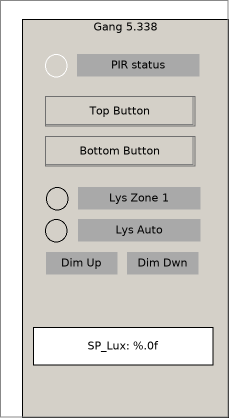
VISUALIZATION Visualization_5_338_1_1  // 229x418
    RoundedRectangle (22,19 207x399), "Gang 5.338"
    Rectangle (33,327 180x38), "SP_Lux: %.0f", text variable: P_Gang_5_338.arrfbLysGruppe[1].fbLightCtrl.fLuxZone1
    Button (45,96 150x30), "Top Button"
        tap P_Gang_5_338.bTopButtonZone1_Visu
    Button (45,136 150x30), "Bottom Button"
        tap P_Gang_5_338.bBottomButtonZone1_Visu
    Ellipse (46,187 22x23), colour toggle: P_Gang_5_338.arrfbLysGruppe[1].fbLightCtrl.bOnZone1
    Rectangle (78,187 122x22), "Lys Zone 1"
    Rectangle (46,252 71x22), "Dim Up", colour toggle: P_Gang_5_338.arrfbLysGruppe[1].fbLightCtrl.bDimUp
    Rectangle (127,252 71x22), "Dim Dwn", colour toggle: P_Gang_5_338.arrfbLysGruppe[1].fbLightCtrl.bDimDwn
    Ellipse (45,219 22x23), colour toggle: P_Gang_5_338.arrfbLysGruppe[1].fbLightCtrl.bAutoZone1
    Rectangle (78,219 122x22), "Lys Auto"
    Ellipse (45,54 22x23), colour toggle: P_Gang_5_338.arrfbLysGruppe[1].fbLightCtrl.bPIR
    Rectangle (77,54 122x22), "PIR status"
END_VISUALIZATION

// ---- POUs/Alle_Rum/Rum_Med_DALI_Pir/Rum_1_435/Visualization_5_338_1_1_1.TcVIS
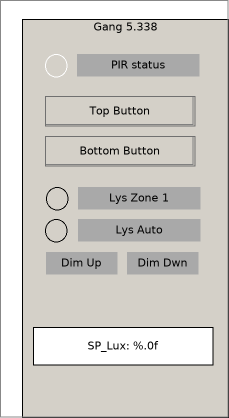
VISUALIZATION Visualization_5_338_1_1_1  // 229x418
    RoundedRectangle (22,19 207x399), "Gang 5.338"
    Rectangle (33,327 180x38), "SP_Lux: %.0f", text variable: P_Gang_5_338.arrfbLysGruppe[1].fbLightCtrl.fLuxZone1
    Button (45,96 150x30), "Top Button"
        tap P_Gang_5_338.bTopButtonZone1_Visu
    Button (45,136 150x30), "Bottom Button"
        tap P_Gang_5_338.bBottomButtonZone1_Visu
    Ellipse (46,187 22x23), colour toggle: P_Gang_5_338.arrfbLysGruppe[1].fbLightCtrl.bOnZone1
    Rectangle (78,187 122x22), "Lys Zone 1"
    Rectangle (46,252 71x22), "Dim Up", colour toggle: P_Gang_5_338.arrfbLysGruppe[1].fbLightCtrl.bDimUp
    Rectangle (127,252 71x22), "Dim Dwn", colour toggle: P_Gang_5_338.arrfbLysGruppe[1].fbLightCtrl.bDimDwn
    Ellipse (45,219 22x23), colour toggle: P_Gang_5_338.arrfbLysGruppe[1].fbLightCtrl.bAutoZone1
    Rectangle (78,219 122x22), "Lys Auto"
    Ellipse (45,54 22x23), colour toggle: P_Gang_5_338.arrfbLysGruppe[1].fbLightCtrl.bPIR
    Rectangle (77,54 122x22), "PIR status"
END_VISUALIZATION

// ---- POUs/Alle_Rum/Rum_Med_DALI_Pir/Rum_1_433/Visualization_5_338_1_1_1_1.TcVIS
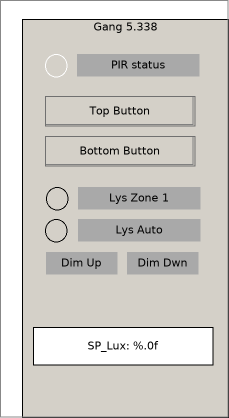
VISUALIZATION Visualization_5_338_1_1_1_1  // 229x418
    RoundedRectangle (22,19 207x399), "Gang 5.338"
    Rectangle (33,327 180x38), "SP_Lux: %.0f", text variable: P_Gang_5_338.arrfbLysGruppe[1].fbLightCtrl.fLuxZone1
    Button (45,96 150x30), "Top Button"
        tap P_Gang_5_338.bTopButtonZone1_Visu
    Button (45,136 150x30), "Bottom Button"
        tap P_Gang_5_338.bBottomButtonZone1_Visu
    Ellipse (46,187 22x23), colour toggle: P_Gang_5_338.arrfbLysGruppe[1].fbLightCtrl.bOnZone1
    Rectangle (78,187 122x22), "Lys Zone 1"
    Rectangle (46,252 71x22), "Dim Up", colour toggle: P_Gang_5_338.arrfbLysGruppe[1].fbLightCtrl.bDimUp
    Rectangle (127,252 71x22), "Dim Dwn", colour toggle: P_Gang_5_338.arrfbLysGruppe[1].fbLightCtrl.bDimDwn
    Ellipse (45,219 22x23), colour toggle: P_Gang_5_338.arrfbLysGruppe[1].fbLightCtrl.bAutoZone1
    Rectangle (78,219 122x22), "Lys Auto"
    Ellipse (45,54 22x23), colour toggle: P_Gang_5_338.arrfbLysGruppe[1].fbLightCtrl.bPIR
    Rectangle (77,54 122x22), "PIR status"
END_VISUALIZATION

// ---- POUs/Alle_Rum/Rum_Med_DALI_Pir/Rum_1_425/Visualization_4_330_1_1_1_1_2_1.TcVIS
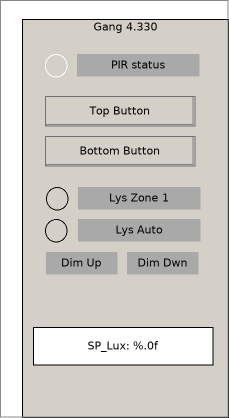
VISUALIZATION Visualization_4_330_1_1_1_1_2_1  // 229x418
    RoundedRectangle (22,19 207x399), "Gang 4.330"
    Rectangle (33,327 180x38), "SP_Lux: %.0f", text variable: P_Gang_5_135A.arrfbLysGruppe[1].fbLightCtrl.fLuxZone1
    Button (45,96 150x30), "Top Button"
        tap P_Gang_5_135A.bTopButtonZone1_Visu
    Button (45,136 150x30), "Bottom Button"
        tap P_Gang_5_135A.bBottomButtonZone1_Visu
    Ellipse (46,187 22x23), colour toggle: P_Gang_5_135A.fbLys.fbLightCtrl.bOnZone1
    Rectangle (78,187 122x22), "Lys Zone 1"
    Rectangle (46,252 71x22), "Dim Up", colour toggle: P_Gang_5_135A.arrfbLysGruppe[1].fbLightCtrl.bDimUp
    Rectangle (127,252 71x22), "Dim Dwn", colour toggle: P_Gang_5_135A.arrfbLysGruppe[1].fbLightCtrl.bDimDwn
    Ellipse (45,219 22x23), colour toggle: P_Gang_5_135A.arrfbLysGruppe[1].fbLightCtrl.bAutoZone1
    Rectangle (78,219 122x22), "Lys Auto"
    Ellipse (45,54 22x23), colour toggle: P_Gang_5_135A.arrfbLysGruppe[1].fbLightCtrl.bPIR
    Rectangle (77,54 122x22), "PIR status"
END_VISUALIZATION

// ---- POUs/DALI/DALI_Setup/VISUs/TextLists/FastFadeTime.TcTLO
TEXTLIST FastFadeTime
  0 = 'Disabled'
  4 = 'T100ms'
  8 = 'T200ms'
  12 = 'T300ms'
  16 = 'T400ms'
  20 = 'T500ms'
  24 = 'T600ms'
  27 = 'T700ms'
  255 = 'Unknown'
   = ''
END_TEXTLIST

// ---- POUs/DALI/DALI_Setup/VISUs/Visu_DALICommissioning.TcVIS
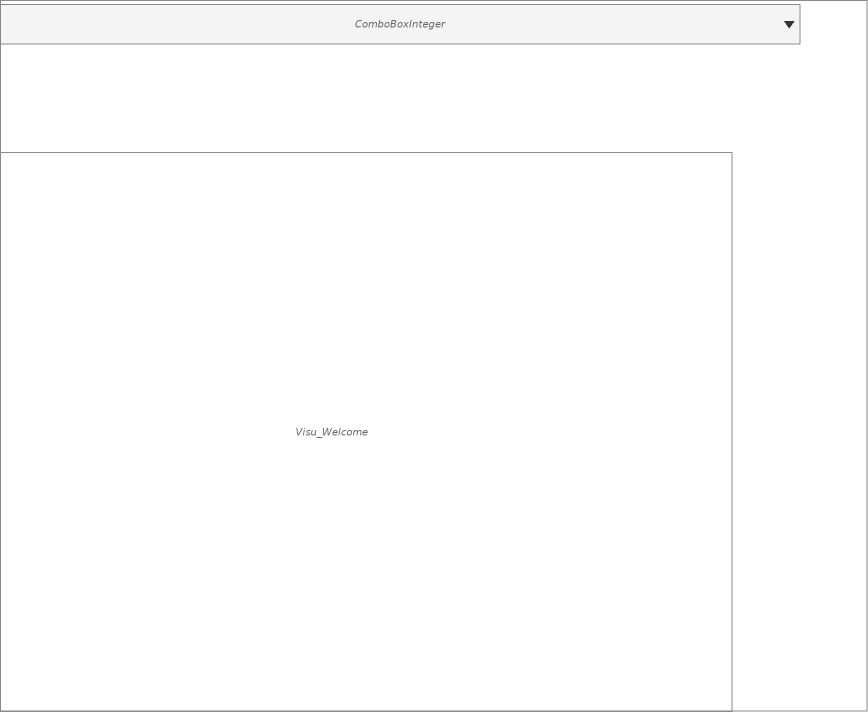
VISUALIZATION Visu_DALICommissioning  // 868x712
    ComboBoxInteger (0,4 800x40), variable: DALI_Commissioning.nSelectedDialog, input disabled if: DALI_Commissioning.bDisableComboBox, text list: 'TextList_Dialogs'
    Frame (-68,152 800x560), frame switch variable: DALI_Commissioning.nSelectedDialog
        shows Visu_Welcome()
        shows Visu_Part102Commands()
        shows Visu_Part102Addressing()
        shows Visu_Part102Parameters()
        shows Visu_Part102Groups()
        shows Visu_Part102Scenes()
        shows Visu_Part102MemoryBank()
        shows Visu_Part102SetFading()
        shows Visu_Part202()
        shows Visu_Part205()
        shows Visu_Part207()
        shows Visu_Part208Switching()
        shows Visu_Part103Addressing()
        shows Visu_Part103Parameters()
        shows Visu_Part103Identify()
        shows Visu_Part301PushButton()
        shows Visu_Part302AbsoluteInputDevice()
        shows Visu_Part303OccupancySensor()
        shows Visu_Part304LightSensor()
        shows Visu_Part300GenericDevice()
        shows Visu_Part103MemoryBank()
        shows Visu_KL6821Configuration()
END_VISUALIZATION

// ---- POUs/DALI/DALI_Setup/VISUs/Visu_DALICommissioning/Visu_Part202Commands.TcVIS
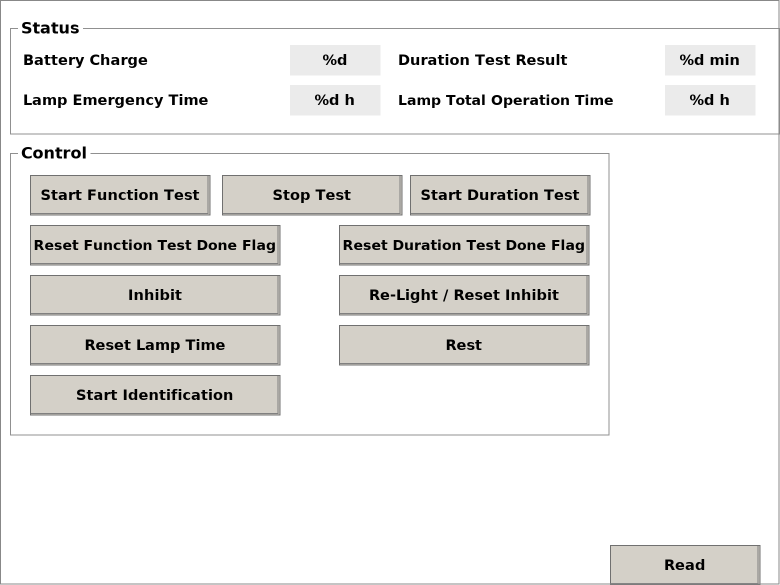
VISUALIZATION Visu_Part202Commands  // 780x585
    GroupBox (10,145 599x290), "Control"
        Button (20,130 250x40), "Inhibit"
            OnMouseClick: execute { DALI_Commissioning.fbPart202Emergency.bInhibit := TRUE; }
        Button (20,80 250x40), "Reset Function Test Done Flag"
            OnMouseClick: execute { DALI_Commissioning.fbPart202Emergency.bResetFunctionTestDoneFlag := TRUE; }
        Button (20,30 180x40), "Start Function Test"
            OnMouseClick: execute { DALI_Commissioning.fbPart202Emergency.bStartFunctionTest := true; }
        Button (20,180 250x40), "Reset Lamp Time"
            OnMouseClick: execute { DALI_Commissioning.fbPart202Emergency.bResetLampTime := TRUE; }
        Button (20,230 250x40), "Start Identification"
            OnMouseClick: execute { DALI_Commissioning.fbPart202Emergency.bStartIdentification := TRUE; }
        Button (212,30 180x40), "Stop Test"
            OnMouseClick: execute { DALI_Commissioning.fbPart202Emergency.bStopTest := TRUE; }
        Button (400,30 180x40), "Start Duration Test"
            OnMouseClick: execute { DALI_Commissioning.fbPart202Emergency.bStartDurationTest := TRUE; }
        Button (329,130 250x40), "Re-Light / Reset Inhibit"
            OnMouseClick: execute { DALI_Commissioning.fbPart202Emergency.bResetInhibit := TRUE; }
    GroupBox (10,20 770x114), "Status"
        Textfield (385,65 220x30), "Lamp Total Operation Time"
        Textfield (655,65 90x30), "%d h", text variable: DALI_Commissioning.fbPart202Emergency.nLampTotalOperationTime
        Textfield (655,25 90x30), "%d min", text variable: DALI_Commissioning.fbPart202Emergency.nDurationTestResult
        Textfield (280,65 90x30), "%d h", text variable: DALI_Commissioning.fbPart202Emergency.nLampEmergencyTime
        Textfield (280,25 90x30), "%d", text variable: DALI_Commissioning.fbPart202Emergency.nBatteryCharge
        Textfield (10,25 220x30), "Battery Charge"
        Textfield (10,65 220x30), "Lamp Emergency Time"
        Textfield (385,25 220x30), "Duration Test Result"
    Button (339,225 250x40), "Reset Duration Test Done Flag"
        OnMouseClick: execute { DALI_Commissioning.fbPart202Emergency.bResetDurationTestDoneFlag := TRUE; }
    Button (339,325 250x40), "Rest"
        OnMouseClick: execute { DALI_Commissioning.fbPart202Emergency.bRest := TRUE; }
    Button (610,545 150x40), "Read"
        OnMouseClick: execute { DALI_Commissioning.fbPart202Emergency.bReadCommands:=TRUE; }
END_VISUALIZATION

// ---- POUs/DALI/DALI_Setup/VISUs/Visu_DALICommissioning/Visu_Part301PushButton.TcVIS
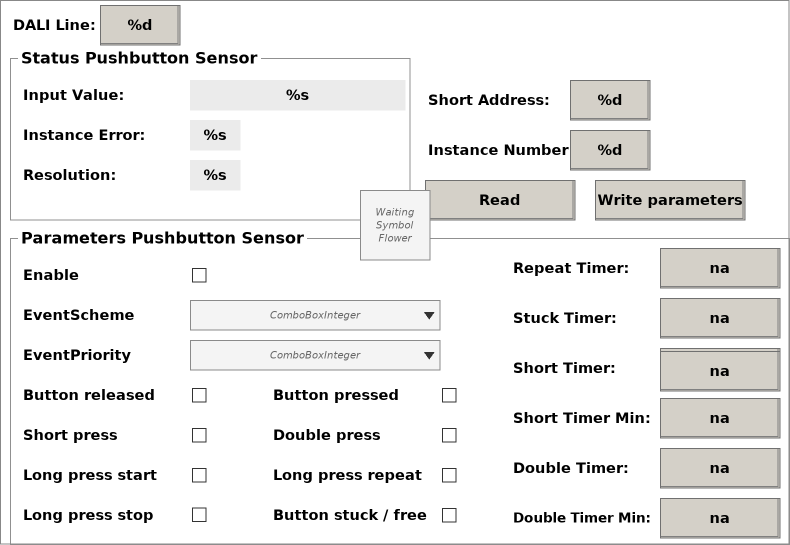
VISUALIZATION Visu_Part301PushButton  // 790x545
    GroupBox (10,230 780x315), "Parameters Pushbutton Sensor"
        Button (650,268 120x40), "%d ms", text variable: DALI_Commissioning.fbPart301PushButton.nDoubleMin
        Button (650,268 120x40), "na", invisible if: Not DALI_Commissioning.fbPart301PushButton.bNoDoubleTimer, input disabled if: Not DALI_Commissioning.fbPart301PushButton.bNoDoubleTimer
        Button (650,168 120x40), "%d ms", text variable: DALI_Commissioning.fbPart301PushButton.nShortMin
        Button (650,168 120x40), "na", invisible if: Not DALI_Commissioning.fbPart301PushButton.bNoRepeatTimer, input disabled if: Not DALI_Commissioning.fbPart301PushButton.bNoRepeatTimer
        Button (650,218 120x40), "%d ms", text variable: DALI_Commissioning.fbPart301PushButton.nDouble
            OnMouseClick: write the text variable via Default, min 0, max 2000, title "Insert value for double timer"
        Button (650,218 120x40), "na", invisible if: Not DALI_Commissioning.fbPart301PushButton.bNoDoubleTimer, input disabled if: Not DALI_Commissioning.fbPart301PushButton.bNoDoubleTimer
        Button (650,118 120x40), "%d ms", text variable: DALI_Commissioning.fbPart301PushButton.nShort
            OnMouseClick: write the text variable via Default, min 10, max 500, title "Insert value for short timer"
        Button (650,121 120x40), "na", invisible if: Not DALI_Commissioning.fbPart301PushButton.bNoRepeatTimer, input disabled if: Not DALI_Commissioning.fbPart301PushButton.bNoRepeatTimer
        Button (650,68 120x40), "%d s", text variable: DALI_Commissioning.fbPart301PushButton.nStuck
            OnMouseClick: write the text variable via Default, min 5, max 255, title "Insert value for stuck timer"
        Button (650,68 120x40), "na", invisible if: Not DALI_Commissioning.fbPart301PushButton.bNoRepeatTimer, input disabled if: Not DALI_Commissioning.fbPart301PushButton.bNoRepeatTimer
        Button (650,18 120x40), "%d ms", text variable: DALI_Commissioning.fbPart301PushButton.nRepeat
            OnMouseClick: write the text variable via Default, min 100, max 2000, title "Insert value for repeat timer"
        Button (650,18 120x40), "na", invisible if: Not DALI_Commissioning.fbPart301PushButton.bNoRepeatTimer, input disabled if: Not DALI_Commissioning.fbPart301PushButton.bNoRepeatTimer
        Textfield (500,23 145x30), "Repeat Timer:"
        Textfield (500,73 145x30), "Stuck Timer:"
        Textfield (500,123 145x30), "Short Timer:"
        Textfield (500,223 145x30), "Double Timer:"
        Textfield (10,30 170x30), "Enable"
        Checkbox (180,30 30x30), variable: DALI_Commissioning.fbPart301PushButton.bEnable
        Textfield (10,70 170x30), "EventScheme"
        Textfield (10,150 170x30), "Button released"
        Textfield (10,190 170x30), "Short press"
        Textfield (10,230 170x30), "Long press start"
        Textfield (10,270 170x30), "Long press stop"
        Textfield (260,150 170x30), "Button pressed"
        Textfield (260,190 170x30), "Double press"
        Textfield (260,230 170x30), "Long press repeat"
        Textfield (260,270 170x30), "Button stuck / free"
        Checkbox (180,150 30x30), variable: DALI_Commissioning.fbPart301PushButton.bButtonReleased
        Checkbox (180,190 30x30), variable: DALI_Commissioning.fbPart301PushButton.bShortPress
        Checkbox (180,230 30x30), variable: DALI_Commissioning.fbPart301PushButton.bLongPressStart
        Checkbox (430,150 30x30), variable: DALI_Commissioning.fbPart301PushButton.bButtonPressed
        Checkbox (430,190 30x30), variable: DALI_Commissioning.fbPart301PushButton.bDoublePress
        Checkbox (430,230 29x30), variable: DALI_Commissioning.fbPart301PushButton.bLongPressRepeat
        Checkbox (430,270 30x30), variable: DALI_Commissioning.fbPart301PushButton.bButtonStuck
        ComboBoxInteger (180,70 250x30), variable: DALI_Commissioning.fbPart301PushButton.eEventScheme, text list: 'EventScheme'
        Checkbox (180,270 28x29), variable: DALI_Commissioning.fbPart301PushButton.bLongPressStop
        Textfield (10,110 170x30), "EventPriority"
        ComboBoxInteger (180,110 250x30), variable: DALI_Commissioning.fbPart301PushButton.eEventPriority, text list: 'EventPriority'
        Textfield (500,173 145x30), "Short Timer Min:"
        Textfield (500,273 145x30), "Double Timer Min:"
    GroupBox (10,50 400x170), "Status Pushbutton Sensor"
        Textfield (10,30 160x30), "Input Value:"
        Textfield (10,70 160x30), "Instance Error:"
        Textfield (10,110 160x30), "Resolution:"
        Textfield (180,30 215x30), "%s", text variable: DALI_Commissioning.fbPart301PushButton.sInputValue
        Textfield (180,70 50x30), "%s", text variable: DALI_Commissioning.fbPart301PushButton.nInstanceError
        Textfield (180,110 50x30), "%s", text variable: DALI_Commissioning.fbPart301PushButton.nResolution
    Button (425,180 150x40), "Read"
        OnMouseClick: execute { DALI_Commissioning.fbPart301PushButton.bRead := TRUE; }
    WaitingSymbolFlower (360,190 70x70), invisible if: DALI_Commissioning.fbPart301PushButton.bHideWaitSymbol
    Button (595,180 150x40), "Write parameters"
        OnMouseClick: execute { DALI_Commissioning.fbPart301PushButton.bWrite := TRUE; }
    Group (10,5 170x40)
        Textfield (0,0 110x40), "DALI Line:"
        Button (90,0 80x40), "%d", text variable: GVL_Internal.nDALILine
            OnMouseClick: write the text variable via Default, min 1, max 10, title "Choose line"
    Textfield (425,80 160x40), "Short Address:"
    Button (570,80 80x40), "%d", text variable: DALI_Commissioning.fbPart301PushButton.nAddress
        OnMouseClick: write the text variable via Default, min 0, max 63, title "Insert Short Address"
    Textfield (425,130 150x40), "Instance Number:"
    Button (570,130 80x40), "%d", text variable: DALI_Commissioning.fbPart301PushButton.nInstanceAddress
        OnMouseClick: write the text variable via Default, min 0, max 31, title "Insert instance number"
END_VISUALIZATION
